// TIA Portal V16 export
// export: Created 2021-11-12T13:31:44.6822865Z, ExportSetting WithDefaults, DisplayName Totally Integrated Automation Portal, DisplayVersion V16 Update 3, DisplayName TIA Portal Version Control Interface, DisplayVersion V16 Update 2, DisplayName TIA Portal Openness, DisplayVersion V16 Update 3, DisplayName SINAMICS Startdrive Advanced, DisplayVersion V16 Update 5, DisplayName SINAMICS Startdrive G130, G150, S120, S150, SINAMICS MV, S210, DisplayVersion V16 Update 5, DisplayName SINAMICS Startdrive G110M, G120, G120C, G120D, G120P, G115D, DisplayVersion V16 Update 5, DisplayName STEP 7 Professional, DisplayVersion V16 Update 3, DisplayName STEP 7 Safety, DisplayVersion V16, DisplayName WinCC UA Professional, DisplayVersion V16 Update 3
FUNCTION "MTS_UpdateTimeInPress" : Void   // FC5, LAD
TITLE = Update time in press machine
{ S7_Optimized_Access := 'TRUE' }
VERSION : 0.1
// Update time in press machine and compare it with technology time limits
// stored: AutoNumber true, IsIECCheckEnabled false, SetENOAutomatically false, UDAEnableTagReadback false
   VAR_INPUT
      IB1Clock_1s : Bool;   // Clock 1 Hz
   END_VAR
   VAR_IN_OUT
      XS_Position : "UDT_MatCard";   // Material data
   END_VAR
   VAR_TEMP
      TB1Enable : Bool;
   END_VAR
BEGIN

REGION Network 1: Enable
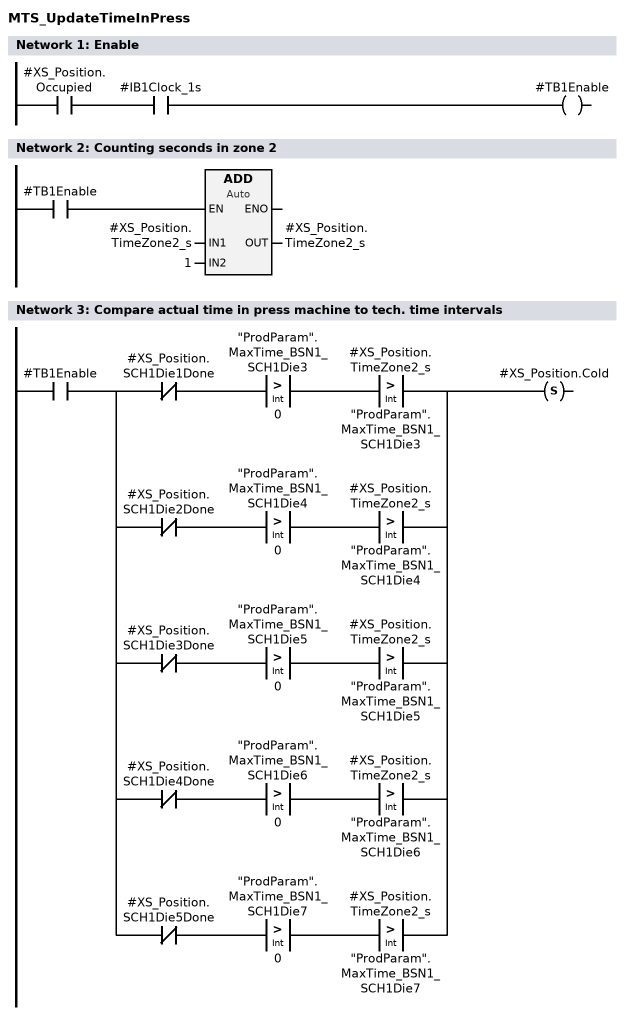
   RUNG wire#powerrail
      Contact( #XS_Position.Occupied )
      Contact( #IB1Clock_1s )
      Coil( #TB1Enable )
   END_RUNG
   // the same network as SCL:
   #TB1Enable := #XS_Position.Occupied AND #IB1Clock_1s;
END_REGION

REGION Network 2: Counting seconds in zone 2
   RUNG wire#powerrail
      Contact( #TB1Enable )
      Add(in1 := #XS_Position.TimeZone2_s, in2 := 1, out => #XS_Position.TimeZone2_s)
   END_RUNG
   // the same network as SCL:
   IF #TB1Enable THEN #XS_Position.TimeZone2_s := #XS_Position.TimeZone2_s + 1; END_IF;
END_REGION

REGION Network 3: Compare actual time in press machine to tech. time intervals
   RUNG wire#powerrail
      Contact( #TB1Enable )
      wire#w1
      I_Contact( #XS_Position.SCH1Die1Done )
      { S7_Templates := "SrcType := Int" } GT_Contact(in1 := "ProdParam".MaxTime_BSN1_SCH1Die3, in2 := 0)
      { S7_Templates := "SrcType := Int" } GT_Contact(in1 := #XS_Position.TimeZone2_s, in2 := "ProdParam".MaxTime_BSN1_SCH1Die3)
      wire#w2
      S_Coil( #XS_Position.Cold )
   END_RUNG
   RUNG wire#w1
      I_Contact( #XS_Position.SCH1Die2Done )
      { S7_Templates := "SrcType := Int" } GT_Contact(in1 := "ProdParam".MaxTime_BSN1_SCH1Die4, in2 := 0)
      { S7_Templates := "SrcType := Int" } GT_Contact(in1 := #XS_Position.TimeZone2_s, in2 := "ProdParam".MaxTime_BSN1_SCH1Die4)
   END_RUNG wire#w2
   RUNG wire#w1
      I_Contact( #XS_Position.SCH1Die3Done )
      { S7_Templates := "SrcType := Int" } GT_Contact(in1 := "ProdParam".MaxTime_BSN1_SCH1Die5, in2 := 0)
      { S7_Templates := "SrcType := Int" } GT_Contact(in1 := #XS_Position.TimeZone2_s, in2 := "ProdParam".MaxTime_BSN1_SCH1Die5)
   END_RUNG wire#w2
   RUNG wire#w1
      I_Contact( #XS_Position.SCH1Die4Done )
      { S7_Templates := "SrcType := Int" } GT_Contact(in1 := "ProdParam".MaxTime_BSN1_SCH1Die6, in2 := 0)
      { S7_Templates := "SrcType := Int" } GT_Contact(in1 := #XS_Position.TimeZone2_s, in2 := "ProdParam".MaxTime_BSN1_SCH1Die6)
   END_RUNG wire#w2
   RUNG wire#w1
      I_Contact( #XS_Position.SCH1Die5Done )
      { S7_Templates := "SrcType := Int" } GT_Contact(in1 := "ProdParam".MaxTime_BSN1_SCH1Die7, in2 := 0)
      { S7_Templates := "SrcType := Int" } GT_Contact(in1 := #XS_Position.TimeZone2_s, in2 := "ProdParam".MaxTime_BSN1_SCH1Die7)
   END_RUNG wire#w2
   // the same network as SCL:
   IF #TB1Enable AND ((NOT #XS_Position.SCH1Die1Done AND ("ProdParam".MaxTime_BSN1_SCH1Die3 > 0) AND (#XS_Position.TimeZone2_s > "ProdParam".MaxTime_BSN1_SCH1Die3)) OR (NOT #XS_Position.SCH1Die2Done AND ("ProdParam".MaxTime_BSN1_SCH1Die4 > 0) AND (#XS_Position.TimeZone2_s > "ProdParam".MaxTime_BSN1_SCH1Die4)) OR (NOT #XS_Position.SCH1Die3Done AND ("ProdParam".MaxTime_BSN1_SCH1Die5 > 0) AND (#XS_Position.TimeZone2_s > "ProdParam".MaxTime_BSN1_SCH1Die5)) OR (NOT #XS_Position.SCH1Die4Done AND ("ProdParam".MaxTime_BSN1_SCH1Die6 > 0) AND (#XS_Position.TimeZone2_s > "ProdParam".MaxTime_BSN1_SCH1Die6)) OR (NOT #XS_Position.SCH1Die5Done AND ("ProdParam".MaxTime_BSN1_SCH1Die7 > 0) AND (#XS_Position.TimeZone2_s > "ProdParam".MaxTime_BSN1_SCH1Die7))) THEN
       #XS_Position.Cold := TRUE;
   END_IF;
END_REGION
END_FUNCTION
